(* CoDeSys 2.3.9.28 project: Lift_Codesys.pro *)
(* Libraries: Standard.lib 27.1.09 16:27:38, Util.lib 27.1.09 16:27:38, IecSfc.lib 24.11.08 13:07:16, SysLibTime.lib 27.1.09 16:27:38, SysTaskInfo.lib 24.11.08 13:07:16, SYSLIBCALLBACK.LIB 27.1.09 16:27:38 *)

(* PLC configuration (modules and I/O channels)
Hexswitch AT %IB0 [HexSwitch] rotary switch 0 = STOP, 1-15 = RUN
AT %IB4 [ByteInput] -
AT %QB0 [ByteOutput] -
AT %IB8 [ByteInput] -
AT %QB4 [ByteOutput] -
*)

(* Global variable list: Global_Variables *)
VAR_GLOBAL
	positieLift : INT;
	stopdeLiftCheck : INT;
	arrayPositie : INT := 0;
	memoryStopAtFloors : ARRAY [1 .. endOfArray] OF INT;
	array_LiftCheck : ARRAY [0 .. endOfArray] OF INT;
	array_positieLift : ARRAY [0 .. endOfArray] OF INT;

	alarmLamp : BOOL;

(*Hulp variabelen*)
	hvBG: BOOL;
	hvBG1: BOOL;
	hvBG2: BOOL;
	hvBG3: BOOL;
	BgAlarm: BOOL;
	hvAlarm : BOOL;


	BgButton:  BOOL;
	Bg1Button: BOOL;
	Bg2Button: BOOL;
	Bg3Button: BOOL;
END_VAR

VAR_GLOBAL CONSTANT
	endOfArray	: INT := 6;
END_VAR

(* POU Hoofdprogramma/PLC_PRG, ST *)
PROGRAM PLC_PRG
VAR
	sensorTrueFalse : BOOL;
	array_Index : INT;
	array_check : INT;
	randomHelp : STRING;
END_VAR
(* Gemaakt door Mohamed Lahmar *)




IF sensorVerdieping1 = TRUE OR sensorVerdieping2 = TRUE OR sensorVerdieping3 = TRUE THEN
	sensorTrueFalse := TRUE;
ELSE
	sensorTrueFalse:= FALSE;
END_IF
END_PROGRAM

(* POU deelPorgrammas/Beveiliging, ST *)
PROGRAM Beveiliging
VAR
	blinker : BLINK;
END_VAR

END_PROGRAM

(* POU deelPorgrammas/Buttons, ST *)
PROGRAM Buttons
VAR
END_VAR

END_PROGRAM

(* POU deelPorgrammas/Sensors, ST *)
PROGRAM Sensors
VAR
	geheugen1 : INT;
END_VAR

END_PROGRAM

(* POU deelPorgrammas/stopLift, ST *)
PROGRAM stopLift
VAR
END_VAR
(* Programma om de lift te stoppen *)

DQ_LiftNaarBeneden := FALSE;
DQ_LiftNaarBoven:= FALSE;

hvBG  := FALSE;
hvBG1 := FALSE;
hvBG2 := FALSE;
hvBG3 := FALSE;
END_PROGRAM

(* Visualisation LIFT
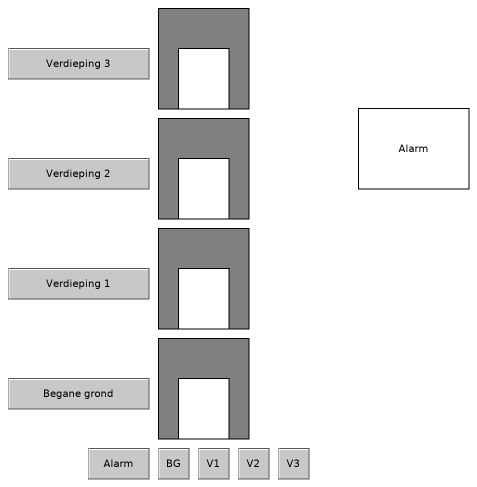
rectangle at (210,340)-(301,441): alarm colour if .eindSensorBeneden
rectangle at (210,230)-(301,331): alarm colour if .sensorVerdieping1
rectangle at (210,120)-(301,221): alarm colour if .sensorVerdieping2
rectangle at (210,10)-(301,111): alarm colour if .sensorVerdieping3
button at (60,380)-(201,411): text "Begane grond"; taps .BgButton
button at (60,270)-(201,301): text "Verdieping 1"; taps .Bg1Button
button at (60,160)-(201,191): text "Verdieping 2"; taps .Bg2Button
button at (60,50)-(201,81): text "Verdieping 3"; taps .Bg3Button
button at (140,450)-(201,481): text "Alarm"; toggles .BgAlarm
button at (210,450)-(241,481): text "BG"; taps .BgButton
button at (250,450)-(281,481): text "V1"; taps .Bg1Button
button at (290,450)-(321,481): text "V2"; taps .Bg2Button
button at (330,450)-(361,481): text "V3"; taps .Bg3Button
rectangle at (410,110)-(521,191): text "Alarm"; alarm colour if .alarmLamp
4 more shapes without text or variables
*)
